{attribute addProperty BoxType "AMP8000-0030-0103-0103"}
{attribute addProperty Id "Std_OutputBIT10.1251Std_OutputBIT10.1252Std_OutputBIT10.1253Std_OutputBIT10.1254Std_OutputBIT10.1255Std_OutputBIT10.1256Std_OutputBIT10.1257Std_OutputBIT10.1258"}
{attribute addProperty CRC "3261648544"}
{attribute addProperty SizeInBites "8"}
{attribute addProperty SizeInBytes "1"}
TYPE FSOE_C268CEA0 :
STRUCT
	{attribute addProperty Name "Std_Output"}
	Std_Output : BIT;
	{attribute addProperty Name "Std_Output"}
	Std_Output_1 : BIT;
	{attribute addProperty Name "Std_Output"}
	Std_Output_2 : BIT;
	{attribute addProperty Name "Std_Output"}
	Std_Output_3 : BIT;
	{attribute addProperty Name "Std_Output"}
	Std_Output_4 : BIT;
	{attribute addProperty Name "Std_Output"}
	Std_Output_5 : BIT;
	{attribute addProperty Name "Std_Output"}
	Std_Output_6 : BIT;
	{attribute addProperty Name "Std_Output"}
	Std_Output_7 : BIT;
END_STRUCT
END_TYPE

(* stored: Version 1.2.0.0, ProductVersion 3.1.4024.9
   DUT FSOE_C268CEA0: Id {ae8879a2-0a31-4341-8ea1-1e878287d90c} *)
